# EPICS substitutions: examples/test/el6002/ecmcEL6002_bytes.substitutions
file "ecmcEcSlave.template"
{
  pattern {}
          {}
}

file "ecmcEL6002-chX_bytes.template"
{
  pattern {CH_ID, PLC_ID, NELM }
          {01,    0,      22   }
          {02,    1,      22   }
}
